PROGRAM MAIN
VAR
	X : INT;
	Y : INT;
END_VAR

END_PROGRAM

(* stored: Version 1.1.0.1, ProductVersion 3.1.4024.12
   POU MAIN: Id {4e1ba2d5-9d55-45b8-9a5c-32eee135143d}, SpecialFunc None *)
